// TIA Portal V15.1 export
// export: Created 2024-06-21T08:40:56.5099425Z, ExportSetting WithDefaults, DisplayName Totally Integrated Automation Portal, DisplayVersion V15.1 Update 5, DisplayName TIA Portal Openness, DisplayVersion V15.1 Update 5, DisplayName SINAMICS Startdrive Advanced, DisplayVersion V15.1, DisplayName G130, G150, S120, S150, SINAMICS MV, S210, DisplayVersion V15.1, DisplayName G110M, G120, G120C, G120D, G120P, DisplayVersion V15.1, DisplayName STEP 7 Professional, DisplayVersion V15.1 Update 5, DisplayName STEP 7 Safety, DisplayVersion V15.1, DisplayName WinCC Professional, DisplayVersion V15.1 Update 5, DisplayName SIMATIC Visualization Architect, DisplayVersion V15.1
FUNCTION_BLOCK "L2StopPos"   // FB1310, FBD
TITLE = L2StopPos
{ S7_Optimized_Access := 'TRUE' }
AUTHOR : VCC
FAMILY : Actuator
VERSION : 0.1
// =============================================================================
// This module will be used for a two Position movements.
// It will take care of the Alarms and of the Detections.
// =============================================================================
// stored: AutoNumber false, IsIECCheckEnabled false, IsRetainMemResEnabled false, MemoryReserve 100, SetENOAutomatically False, UDAEnableTagReadback false
   VAR_INPUT
      I_DetSet { ExternalAccessible := 'False'; ExternalVisible := 'False'; ExternalWritable := 'False'} : Bool;   // Set detection signal / Set Detection signal
      I_DetRes { ExternalAccessible := 'False'; ExternalVisible := 'False'; ExternalWritable := 'False'} : Bool;   // Reset detection signal / Reset Detection signal
      I_CmdSet { ExternalAccessible := 'False'; ExternalVisible := 'False'; ExternalWritable := 'False'} : Bool;   // function set command / Function set command
      I_CmdRes { ExternalAccessible := 'False'; ExternalVisible := 'False'; ExternalWritable := 'False'} : Bool;   // Function reset command / Function Reset command
      I_RunSet { ExternalAccessible := 'False'; ExternalVisible := 'False'; ExternalWritable := 'False'} : Bool;   // Memory that the Set function is busy
      I_RunRes { ExternalAccessible := 'False'; ExternalVisible := 'False'; ExternalWritable := 'False'} : Bool;   // Memory that the Reset function is busy
      I_SetIntlkOK { ExternalAccessible := 'False'; ExternalVisible := 'False'; ExternalWritable := 'False'} : Bool := TRUE;   // Set Interlock
      I_ResIntlkOK { ExternalAccessible := 'False'; ExternalVisible := 'False'; ExternalWritable := 'False'} : Bool := TRUE;   // Reset Interlock
      I_SafetyOk { ExternalAccessible := 'False'; ExternalVisible := 'False'; ExternalWritable := 'False'} : Bool;   // Safety Ok
      I_AlarmResetPB { ExternalAccessible := 'False'; ExternalVisible := 'False'; ExternalWritable := 'False'} : Bool := TRUE;   // alarm reset Push Button is activated / Alarm Reset Push Button is Activated
      C_KeepPosition { ExternalAccessible := 'False'; ExternalVisible := 'False'; ExternalWritable := 'False'} : Bool;   // If true, the last position shall be kept ON and checked / If true, the last Position shall be kept ON and checked
      C_EnAlmDet { ExternalAccessible := 'False'; ExternalVisible := 'False'; ExternalWritable := 'False'} : Bool;   // Enable alarm / Enable Alarm
      C_AlarmResetUsed { ExternalAccessible := 'False'; ExternalVisible := 'False'; ExternalWritable := 'False'} : Bool;   // If true, the alarms will be stored untill reseted / If true, the Alarms will be stored untill Reseted
      C_EnAlmOvertime { ExternalAccessible := 'False'; ExternalVisible := 'False'; ExternalWritable := 'False'} : Bool := TRUE;   // Enable Overtime Alarm
      C_ManualClampCmdSet { ExternalAccessible := 'False'; ExternalVisible := 'False'; ExternalWritable := 'False'} : Bool;   // Manual Clamp Set
      C_ManualClampCmdRes { ExternalAccessible := 'False'; ExternalVisible := 'False'; ExternalWritable := 'False'} : Bool;   // Manual Clamp Reset
      C_RunTimeMaxSetWarn { ExternalAccessible := 'False'; ExternalVisible := 'False'; ExternalWritable := 'False'} : DInt;   // Maximum Time (ms) that the function may run (create overtime) / Maximum Time (ms) that the function may run (create Overtime)
      C_RunTimeMaxSetAlm { ExternalAccessible := 'False'; ExternalVisible := 'False'; ExternalWritable := 'False'} : DInt;   // Maximum Time (ms) that the function may run (create overtime) / Maximum Time (ms) that the function may run (create Overtime)
      C_RunTimeMaxResWarn { ExternalAccessible := 'False'; ExternalVisible := 'False'; ExternalWritable := 'False'} : DInt;   // Maximum Time (ms) that the function may run (create overtime) / Maximum Time (ms) that the function may run (create Overtime)
      C_RunTimeMaxResAlm { ExternalAccessible := 'False'; ExternalVisible := 'False'; ExternalWritable := 'False'} : DInt;   // Maximum Time (ms) that the function may run (create overtime) / Maximum Time (ms) that the function may run (create Overtime)
      C_TimeAlmFilt { ExternalAccessible := 'False'; ExternalVisible := 'False'; ExternalWritable := 'False'} : DInt := L#2000;   // timer before any actuator alarm will be active (welding..) / timer before any actuator Alarm will be active (welding..)
      C_AlarmSeverityAB { ExternalAccessible := 'False'; ExternalVisible := 'False'; ExternalWritable := 'False'} : Bool;   // Alarm severity
      C_RunTimeCalculated { ExternalAccessible := 'False'; ExternalVisible := 'False'; ExternalWritable := 'False'} : Bool;   // Maximum Time (ms) that the function may run (create Overtime) is calculated
   END_VAR
   VAR_OUTPUT
      O_SetPos { ExternalAccessible := 'False'; ExternalVisible := 'False'; ExternalWritable := 'False'} : Bool;   // Actuator is in set position / Actuator is in set Position
      O_ResPos { ExternalAccessible := 'False'; ExternalVisible := 'False'; ExternalWritable := 'False'} : Bool;   // Actuator is in reset position / Actuator is in Reset Position
      O_KeepPosSetAlm { ExternalAccessible := 'False'; ExternalVisible := 'False'; ExternalWritable := 'False'} : Bool;   // Detection Set alarm / Detection Set Alarm
      O_KeepPosResAlm { ExternalAccessible := 'False'; ExternalVisible := 'False'; ExternalWritable := 'False'} : Bool;   // Detection Reset alarm / Detection Reset Alarm
      O_TwoDetAlm { ExternalAccessible := 'False'; ExternalVisible := 'False'; ExternalWritable := 'False'} : Bool;   // Fault condition Both detections ON at the same time
      O_OvtSetWarn { ExternalAccessible := 'False'; ExternalVisible := 'False'; ExternalWritable := 'False'} : Bool;   // Warning Overtime Set
      O_OvtResWarn { ExternalAccessible := 'False'; ExternalVisible := 'False'; ExternalWritable := 'False'} : Bool;   // Warning Overtime Reset
      O_OvtSetAlm { ExternalAccessible := 'False'; ExternalVisible := 'False'; ExternalWritable := 'False'} : Bool;   // Alarm Overtime Set
      O_OvtResAlm { ExternalAccessible := 'False'; ExternalVisible := 'False'; ExternalWritable := 'False'} : Bool;   // Alarm Overtime Reset
      O_ConfigCalibrationAlm { ExternalAccessible := 'False'; ExternalVisible := 'False'; ExternalWritable := 'False'} : Bool;   // Alarm Config/Calibration
      O_CalibrationWarn { ExternalAccessible := 'False'; ExternalVisible := 'False'; ExternalWritable := 'False'} : Bool;   // Warning Calibration
      O_AlarmABCondition { ExternalAccessible := 'False'; ExternalVisible := 'False'; ExternalWritable := 'False'} : Bool;   // Alarm AB condition / Alarm AB Condition
      H_IAnim { ExternalAccessible := 'False'; ExternalVisible := 'False'; ExternalWritable := 'False'} : DWord;   // Animation color of icon
   END_VAR
   VAR_IN_OUT
      IO_Modes : "Modes";   // Modes
      H_2StopPos : "H_2StopPos";   // Animation
   END_VAR
   VAR
      AlarmReset { ExternalAccessible := 'False'; ExternalVisible := 'False'; ExternalWritable := 'False'} : Bool;   // Alarm Reset Memory
      SetPosReq { ExternalAccessible := 'False'; ExternalVisible := 'False'; ExternalWritable := 'False'} : Bool;   // Memorisation of the last set movement
      ResPosReq { ExternalAccessible := 'False'; ExternalVisible := 'False'; ExternalWritable := 'False'} : Bool;   // Memorisation of the last reset movement / Memorisation of the last Reset movement
      KeepSetPosOn { ExternalAccessible := 'False'; ExternalVisible := 'False'; ExternalWritable := 'False'} : Bool;   // Check that Set detection is keept on / Check that Set Detection is keept on
      KeepResPosOn { ExternalAccessible := 'False'; ExternalVisible := 'False'; ExternalWritable := 'False'} : Bool;   // Check that Set detection is keept on / Check that Set Detection is keept on
      KeepPosSetStartTimer { ExternalAccessible := 'False'; ExternalVisible := 'False'; ExternalWritable := 'False'} : Bool;   // Detection Set request to start timer / Detection Set Request to start timer
      KeepPosResStartTimer { ExternalAccessible := 'False'; ExternalVisible := 'False'; ExternalWritable := 'False'} : Bool;   // Detection Reset request to start timer / Detection Reset Request to start timer
      TwoDetStartTimer { ExternalAccessible := 'False'; ExternalVisible := 'False'; ExternalWritable := 'False'} : Bool;   // Both detections ON at the same time request to start timer / Both Detections ON at the same time Request to start timer
      AlarmFilterStart { ExternalAccessible := 'False'; ExternalVisible := 'False'; ExternalWritable := 'False'} : Bool;   // Alarm filter must be started
      OvtSetWarnResult { ExternalAccessible := 'False'; ExternalVisible := 'False'; ExternalWritable := 'False'} : Bool;   // Overtime set warning result
      OvtResWarnResult { ExternalAccessible := 'False'; ExternalVisible := 'False'; ExternalWritable := 'False'} : Bool;   // Overtime reset warning result / Overtime Reset warning result
      OvtSetAlmResult { ExternalAccessible := 'False'; ExternalVisible := 'False'; ExternalWritable := 'False'} : Bool;   // Overtime set alarm result / Overtime set Alarm result
      OvtResAlmResult { ExternalAccessible := 'False'; ExternalVisible := 'False'; ExternalWritable := 'False'} : Bool;   // Overtime reset alarm result / Overtime Reset Alarm result
      AlmFilterResult { ExternalAccessible := 'False'; ExternalVisible := 'False'; ExternalWritable := 'False'} : Bool;   // Alarm filter result
      TwoDetAlm { ExternalAccessible := 'False'; ExternalVisible := 'False'; ExternalWritable := 'False'} : Bool;   // Two detection alarm / Set Reset Activated Simultaneously / Set Reset Påverkade Samtidigt
      KeepPosResAlm { ExternalAccessible := 'False'; ExternalVisible := 'False'; ExternalWritable := 'False'} : Bool;   // Keep position Reset alarm / Position Supervision Reset Position / Positionsövervakning Reset Läge
      KeepPosSetAlm { ExternalAccessible := 'False'; ExternalVisible := 'False'; ExternalWritable := 'False'} : Bool;   // Keep position Set alarm / Alarm Keep Position Set Position / Larm Positionsövervakning Set Läge
      OvtResAlm { ExternalAccessible := 'False'; ExternalVisible := 'False'; ExternalWritable := 'False'} : Bool;   // Overtime Reset alarm / Overtime Reset Alarm
      OvtSetAlm { ExternalAccessible := 'False'; ExternalVisible := 'False'; ExternalWritable := 'False'} : Bool;   // Overtime Set alarm / Timeout Set / Tidsövervakning Set
      OvtResWarn { ExternalAccessible := 'False'; ExternalVisible := 'False'; ExternalWritable := 'False'} : Bool;   // Overtime Reset warning
      OvtSetWarn { ExternalAccessible := 'False'; ExternalVisible := 'False'; ExternalWritable := 'False'} : Bool;   // Overtime Set warning
      ConfigCalibrationAlm { ExternalAccessible := 'False'; ExternalVisible := 'False'; ExternalWritable := 'False'} : Bool;   // Config/Calibration Alarm
      CalibrationWarn { ExternalAccessible := 'False'; ExternalVisible := 'False'; ExternalWritable := 'False'} : Bool;   // Warning Calibration
      SetPos { ExternalAccessible := 'False'; ExternalVisible := 'False'; ExternalWritable := 'False'} : Bool;   // Set position / Set Position
      ResPos { ExternalAccessible := 'False'; ExternalVisible := 'False'; ExternalWritable := 'False'} : Bool;   // Reset position / Reset Position
      KeepPosResAlmCond { ExternalAccessible := 'False'; ExternalVisible := 'False'; ExternalWritable := 'False'} : Bool;   // Keep position reset alarm condition / Keep Position Reset Alarm condition
      KeepPosSetAlmCond { ExternalAccessible := 'False'; ExternalVisible := 'False'; ExternalWritable := 'False'} : Bool;   // Keep position set alarm condition / Keep Position Set Alarm condition
      TwoDetAlmCond { ExternalAccessible := 'False'; ExternalVisible := 'False'; ExternalWritable := 'False'} : Bool;   // Two detector alarm condition / Two detector Alarm condition
      OvtResAlmCond { ExternalAccessible := 'False'; ExternalVisible := 'False'; ExternalWritable := 'False'} : Bool;   // Overtime reset alarm condition / Overtime Reset Alarm condition
      OvtSetAlmCond { ExternalAccessible := 'False'; ExternalVisible := 'False'; ExternalWritable := 'False'} : Bool;   // Overtime set alarm condition / Overtime set Alarm condition
      RunSet { ExternalAccessible := 'False'; ExternalVisible := 'False'; ExternalWritable := 'False'} : Bool;   // Memory that the Set function is busy
      RunRes { ExternalAccessible := 'False'; ExternalVisible := 'False'; ExternalWritable := 'False'} : Bool;   // Memory that the Reset function is busy
      Edge { ExternalAccessible := 'False'; ExternalVisible := 'False'; ExternalWritable := 'False'} : Array[1..8] of Bool;   // Edge
      AlarmTimer { ExternalAccessible := 'False'; ExternalVisible := 'False'; ExternalWritable := 'False'} : "LTimer";   // FB
      OvtSetWarnTimer { ExternalAccessible := 'False'; ExternalVisible := 'False'; ExternalWritable := 'False'} : "LTimer";   // FB
      OvtResWarnTimer { ExternalAccessible := 'False'; ExternalVisible := 'False'; ExternalWritable := 'False'} : "LTimer";   // FB
      OvtSetAlmTimer { ExternalAccessible := 'False'; ExternalVisible := 'False'; ExternalWritable := 'False'} : "LTimer";   // FB
      OvtResAlmTimer { ExternalAccessible := 'False'; ExternalVisible := 'False'; ExternalWritable := 'False'} : "LTimer";   // FB
   END_VAR
   VAR RETAIN
      OvtWarnSet { ExternalAccessible := 'False'; ExternalVisible := 'False'; ExternalWritable := 'False'} : DInt;   // Alarm Value
      OvtWarnRes { ExternalAccessible := 'False'; ExternalVisible := 'False'; ExternalWritable := 'False'} : DInt;   // Alarm Value
      OvtAlarmSet { ExternalAccessible := 'False'; ExternalVisible := 'False'; ExternalWritable := 'False'} : DInt;   // Alarm Value
      OvtAlarmRes { ExternalAccessible := 'False'; ExternalVisible := 'False'; ExternalWritable := 'False'} : DInt;   // Alarm Value
      CalibratedSet { ExternalAccessible := 'False'; ExternalVisible := 'False'; ExternalWritable := 'False'} : Bool;   // Calibrated Set
      CalibratedRes { ExternalAccessible := 'False'; ExternalVisible := 'False'; ExternalWritable := 'False'} : Bool;   // Calibrated Reset
   END_VAR
   VAR
      AlarmTimeWithConfig { ExternalAccessible := 'False'; ExternalVisible := 'False'; ExternalWritable := 'False'} : Bool;
      AlarmTimeWithCalibration { ExternalAccessible := 'False'; ExternalVisible := 'False'; ExternalWritable := 'False'} : Bool;
      AlarmTimeWithCalculation { ExternalAccessible := 'False'; ExternalVisible := 'False'; ExternalWritable := 'False'} : Bool;
      AlmFilterTimerValue { ExternalAccessible := 'False'; ExternalVisible := 'False'; ExternalWritable := 'False'} : DInt;
   END_VAR
   VAR_TEMP
      H_CalibrateSet : Bool;   // HMI Function
      H_CalibrateReset : Bool;   // HMI Function
      TempReal : Real;
   END_VAR
   VAR_TEMP   // added for the SCL form of the ladder/FBD networks
      _w1 : Bool;
      _w2 : Bool;
      _w3 : Bool;
      _w4 : Bool;
   END_VAR
BEGIN

REGION Network 1: **** 1 - Inputs **** HMI Commands
   // Extract the Commands from HMIRobCmd / Extract the Commands from HMI
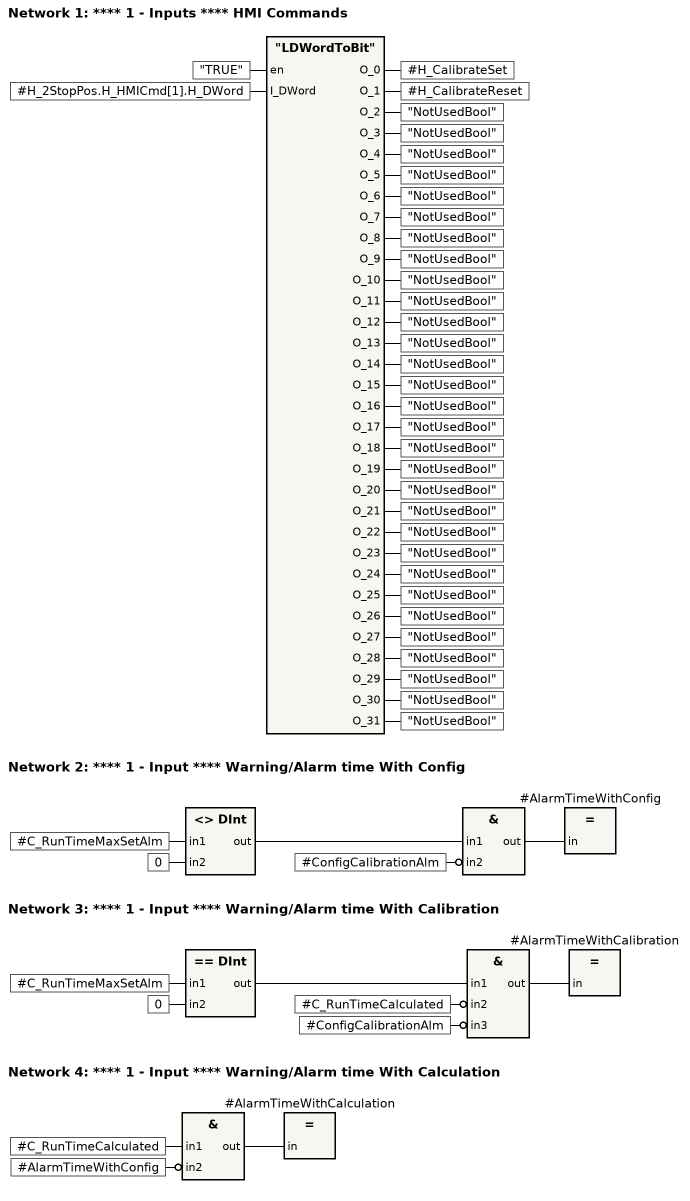
   IF "TRUE" THEN
       "LDWordToBit"(I_DWord := #H_2StopPos.H_HMICmd[1].H_DWord,
                     O_0 => #H_CalibrateSet,
                     O_1 => #H_CalibrateReset,
                     O_2 => "NotUsedBool",
                     O_3 => "NotUsedBool",
                     O_4 => "NotUsedBool",
                     O_5 => "NotUsedBool",
                     O_6 => "NotUsedBool",
                     O_7 => "NotUsedBool",
                     O_8 => "NotUsedBool",
                     O_9 => "NotUsedBool",
                     O_10 => "NotUsedBool",
                     O_11 => "NotUsedBool",
                     O_12 => "NotUsedBool",
                     O_13 => "NotUsedBool",
                     O_14 => "NotUsedBool",
                     O_15 => "NotUsedBool",
                     O_16 => "NotUsedBool",
                     O_17 => "NotUsedBool",
                     O_18 => "NotUsedBool",
                     O_19 => "NotUsedBool",
                     O_20 => "NotUsedBool",
                     O_21 => "NotUsedBool",
                     O_22 => "NotUsedBool",
                     O_23 => "NotUsedBool",
                     O_24 => "NotUsedBool",
                     O_25 => "NotUsedBool",
                     O_26 => "NotUsedBool",
                     O_27 => "NotUsedBool",
                     O_28 => "NotUsedBool",
                     O_29 => "NotUsedBool",
                     O_30 => "NotUsedBool",
                     O_31 => "NotUsedBool");
   END_IF;
END_REGION

REGION Network 2: **** 1 - Input **** Warning/Alarm time With Config
   #AlarmTimeWithConfig := (#C_RunTimeMaxSetAlm <> 0) AND NOT #ConfigCalibrationAlm;
END_REGION

REGION Network 3: **** 1 - Input **** Warning/Alarm time With Calibration
   #AlarmTimeWithCalibration := (#C_RunTimeMaxSetAlm = 0) AND NOT #C_RunTimeCalculated AND NOT #ConfigCalibrationAlm;
END_REGION

REGION Network 4: **** 1 - Input **** Warning/Alarm time With Calculation
   #AlarmTimeWithCalculation := #C_RunTimeCalculated AND NOT #AlarmTimeWithConfig;
END_REGION

REGION Network 5: Calibrated Set / **** 1 - Input **** Ovt Values / **** 1 - Inputs **** Ovt Values
   // Ovt Values
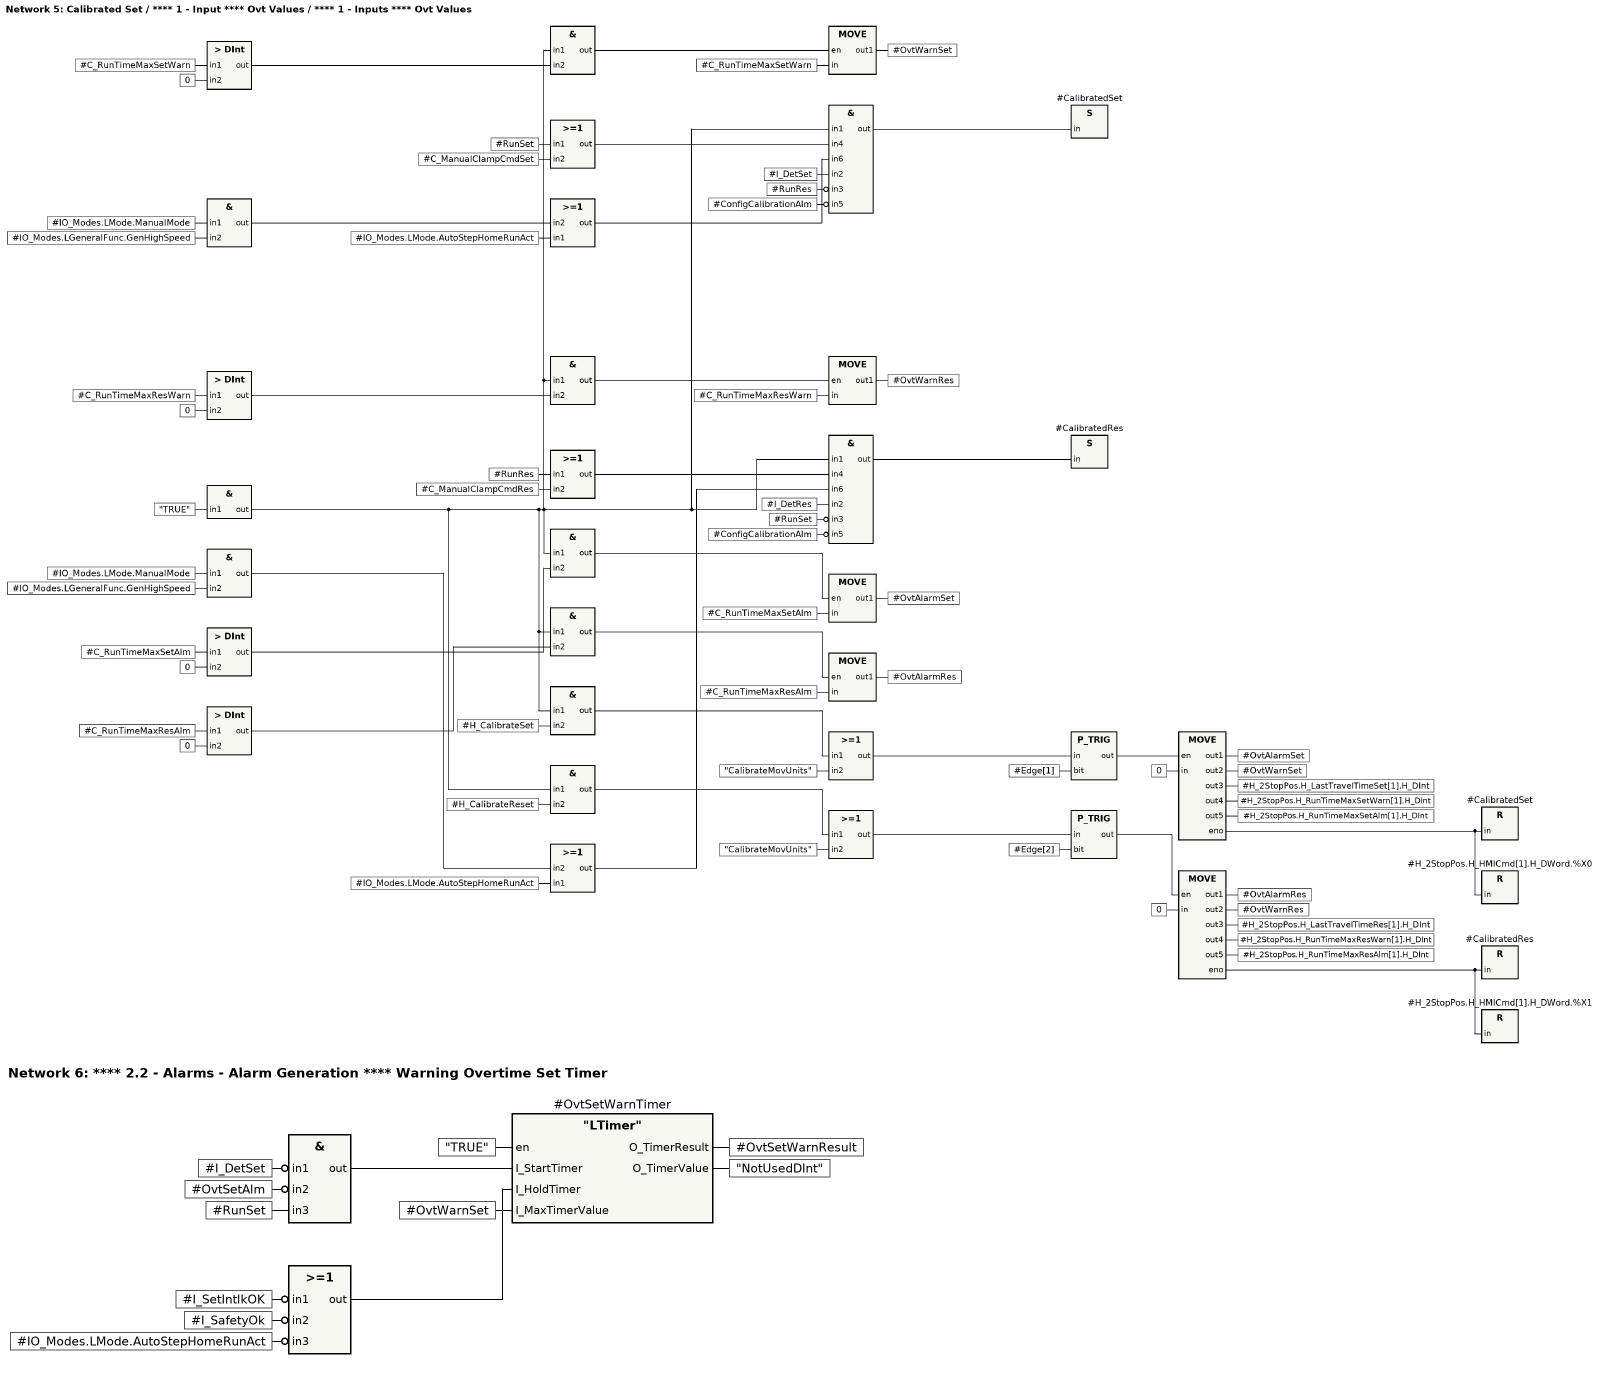
   // ENO of a box is taken as its EN; it also drops when the box reports an error
   IF "TRUE" AND (#C_RunTimeMaxSetWarn > 0) THEN #OvtWarnSet := #C_RunTimeMaxSetWarn; END_IF;
   IF "TRUE" AND (#C_RunTimeMaxResWarn > 0) THEN #OvtWarnRes := #C_RunTimeMaxResWarn; END_IF;
   IF "TRUE" AND (#C_RunTimeMaxSetAlm > 0) THEN #OvtAlarmSet := #C_RunTimeMaxSetAlm; END_IF;
   IF "TRUE" AND (#C_RunTimeMaxResAlm > 0) THEN #OvtAlarmRes := #C_RunTimeMaxResAlm; END_IF;
   IF "TRUE" AND (#RunSet OR #C_ManualClampCmdSet) AND ((#IO_Modes.LMode.ManualMode AND #IO_Modes.LGeneralFunc.GenHighSpeed) OR #IO_Modes.LMode.AutoStepHomeRunAct) AND #I_DetSet AND NOT #RunRes AND NOT #ConfigCalibrationAlm THEN
       #CalibratedSet := TRUE;
   END_IF;
   IF "TRUE" AND (#RunRes OR #C_ManualClampCmdRes) AND ((#IO_Modes.LMode.ManualMode AND #IO_Modes.LGeneralFunc.GenHighSpeed) OR #IO_Modes.LMode.AutoStepHomeRunAct) AND #I_DetRes AND NOT #RunSet AND NOT #ConfigCalibrationAlm THEN
       #CalibratedRes := TRUE;
   END_IF;
   #_w1 := ("TRUE" AND #H_CalibrateSet) OR "CalibrateMovUnits";
   #_w2 := #_w1 AND NOT #Edge[1];   // rising edge
   #Edge[1] := #_w1;
   IF #_w2 THEN
       #OvtAlarmSet := 0;
       #OvtWarnSet := 0;
       #H_2StopPos.H_LastTravelTimeSet[1].H_DInt := 0;
       #H_2StopPos.H_RunTimeMaxSetWarn[1].H_DInt := 0;
       #H_2StopPos.H_RunTimeMaxSetAlm[1].H_DInt := 0;
       #CalibratedSet := FALSE;
       #H_2StopPos.H_HMICmd[1].H_DWord.%X0 := FALSE;
   END_IF;
   #_w3 := ("TRUE" AND #H_CalibrateReset) OR "CalibrateMovUnits";
   #_w4 := #_w3 AND NOT #Edge[2];   // rising edge
   #Edge[2] := #_w3;
   IF #_w4 THEN
       #OvtAlarmRes := 0;
       #OvtWarnRes := 0;
       #H_2StopPos.H_LastTravelTimeRes[1].H_DInt := 0;
       #H_2StopPos.H_RunTimeMaxResWarn[1].H_DInt := 0;
       #H_2StopPos.H_RunTimeMaxResAlm[1].H_DInt := 0;
       #CalibratedRes := FALSE;
       #H_2StopPos.H_HMICmd[1].H_DWord.%X1 := FALSE;
   END_IF;
END_REGION

REGION Network 6: **** 2.2 - Alarms - Alarm Generation **** Warning Overtime Set Timer
   // Warning Overtime Set Timer
   IF "TRUE" THEN
       #OvtSetWarnTimer(I_StartTimer := NOT #I_DetSet AND NOT #OvtSetAlm AND #RunSet,   // "LTimer"
                        I_HoldTimer := NOT #I_SetIntlkOK OR NOT #I_SafetyOk OR NOT #IO_Modes.LMode.AutoStepHomeRunAct,
                        I_MaxTimerValue := #OvtWarnSet,
                        O_TimerResult => #OvtSetWarnResult,
                        O_TimerValue => "NotUsedDInt");
   END_IF;
END_REGION

REGION Network 7: **** 2.2 - Alarms - Alarm Generation **** Warning Overtime Set Memorisation
   // Warning Overtime Set Memorisation
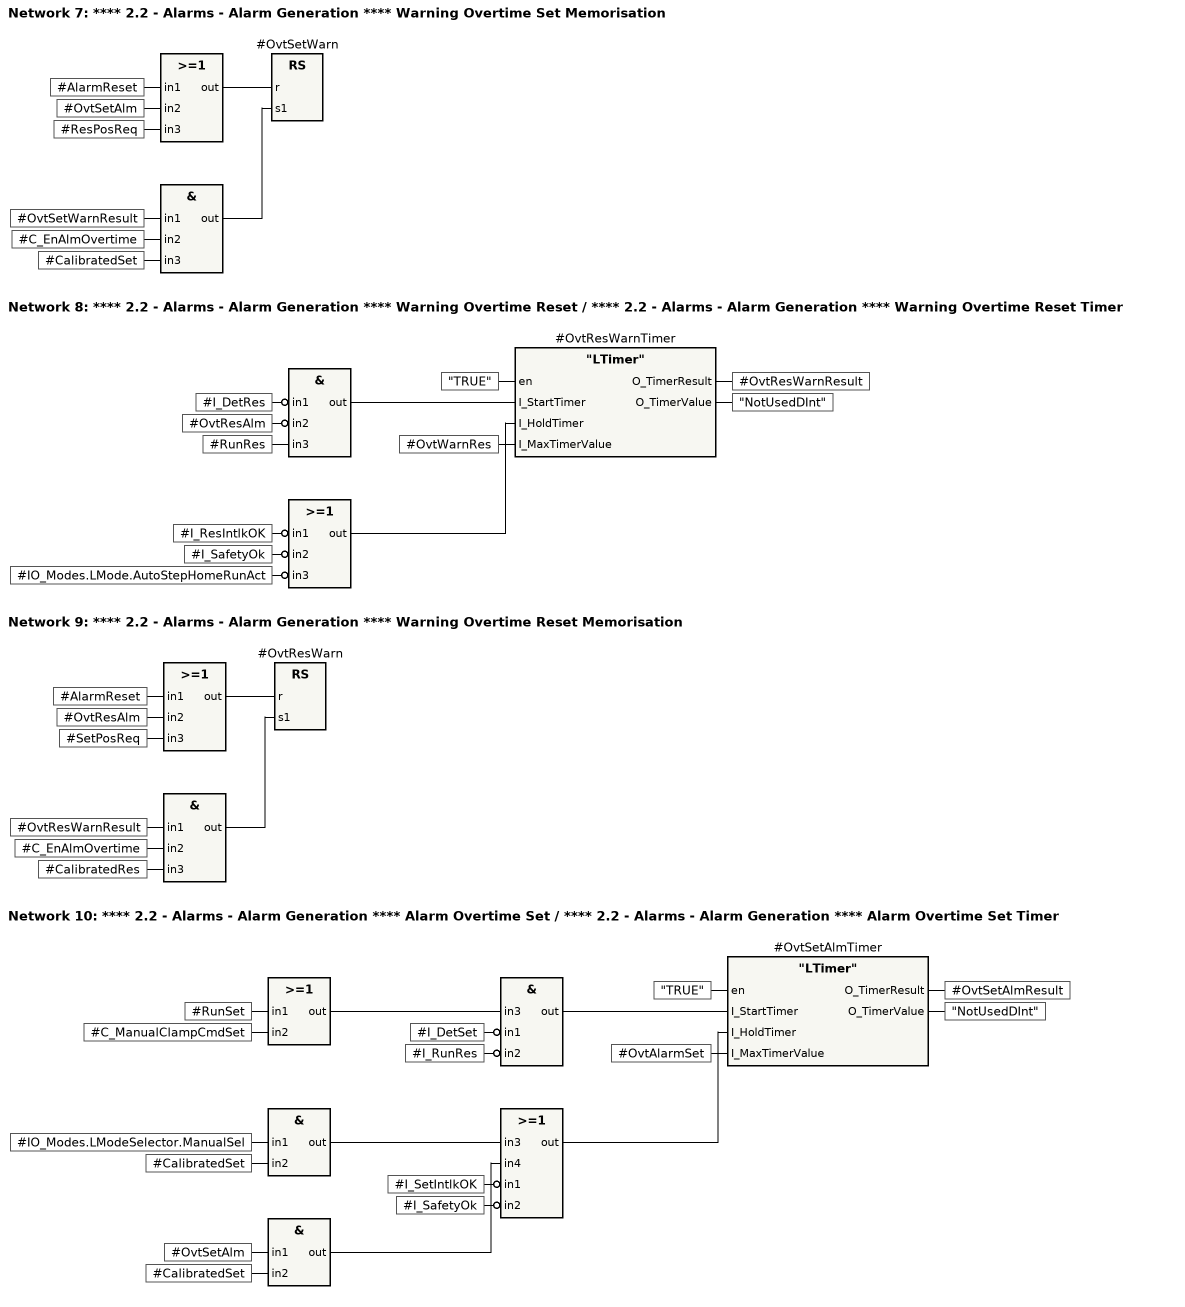
   IF #AlarmReset OR #OvtSetAlm OR #ResPosReq THEN
       #OvtSetWarn := FALSE;   // RS flip-flop
   END_IF;
   IF #OvtSetWarnResult AND #C_EnAlmOvertime AND #CalibratedSet THEN #OvtSetWarn := TRUE; END_IF;
END_REGION

REGION Network 8: **** 2.2 - Alarms - Alarm Generation **** Warning Overtime Reset / **** 2.2 - Alarms - Alarm Generation **** Warning Overtime Reset Timer
   // Warning Overtime Reset
   IF "TRUE" THEN
       #OvtResWarnTimer(I_StartTimer := NOT #I_DetRes AND NOT #OvtResAlm AND #RunRes,   // "LTimer"
                        I_HoldTimer := NOT #I_ResIntlkOK OR NOT #I_SafetyOk OR NOT #IO_Modes.LMode.AutoStepHomeRunAct,
                        I_MaxTimerValue := #OvtWarnRes,
                        O_TimerResult => #OvtResWarnResult,
                        O_TimerValue => "NotUsedDInt");
   END_IF;
END_REGION

REGION Network 9: **** 2.2 - Alarms - Alarm Generation **** Warning Overtime Reset Memorisation
   // Warning Overtime Reset  Memorisation
   IF #AlarmReset OR #OvtResAlm OR #SetPosReq THEN
       #OvtResWarn := FALSE;   // RS flip-flop
   END_IF;
   IF #OvtResWarnResult AND #C_EnAlmOvertime AND #CalibratedRes THEN #OvtResWarn := TRUE; END_IF;
END_REGION

REGION Network 10: **** 2.2 - Alarms - Alarm Generation **** Alarm Overtime Set / **** 2.2 - Alarms - Alarm Generation **** Alarm Overtime Set Timer
   // Alarm Overtime Set
   IF "TRUE" THEN
       #OvtSetAlmTimer(I_StartTimer := (#RunSet OR #C_ManualClampCmdSet) AND NOT #I_DetSet AND NOT #I_RunRes,   // "LTimer"
                       I_HoldTimer := (#IO_Modes.LModeSelector.ManualSel AND #CalibratedSet) OR (#OvtSetAlm AND #CalibratedSet) OR NOT #I_SetIntlkOK OR NOT #I_SafetyOk,
                       I_MaxTimerValue := #OvtAlarmSet,
                       O_TimerResult => #OvtSetAlmResult,
                       O_TimerValue => "NotUsedDInt");
   END_IF;
END_REGION

REGION Network 11: **** 2.2 - Alarms - Alarm Generation **** Alarm Overtime Set Timer -- Calculation Warning/Alarm Time
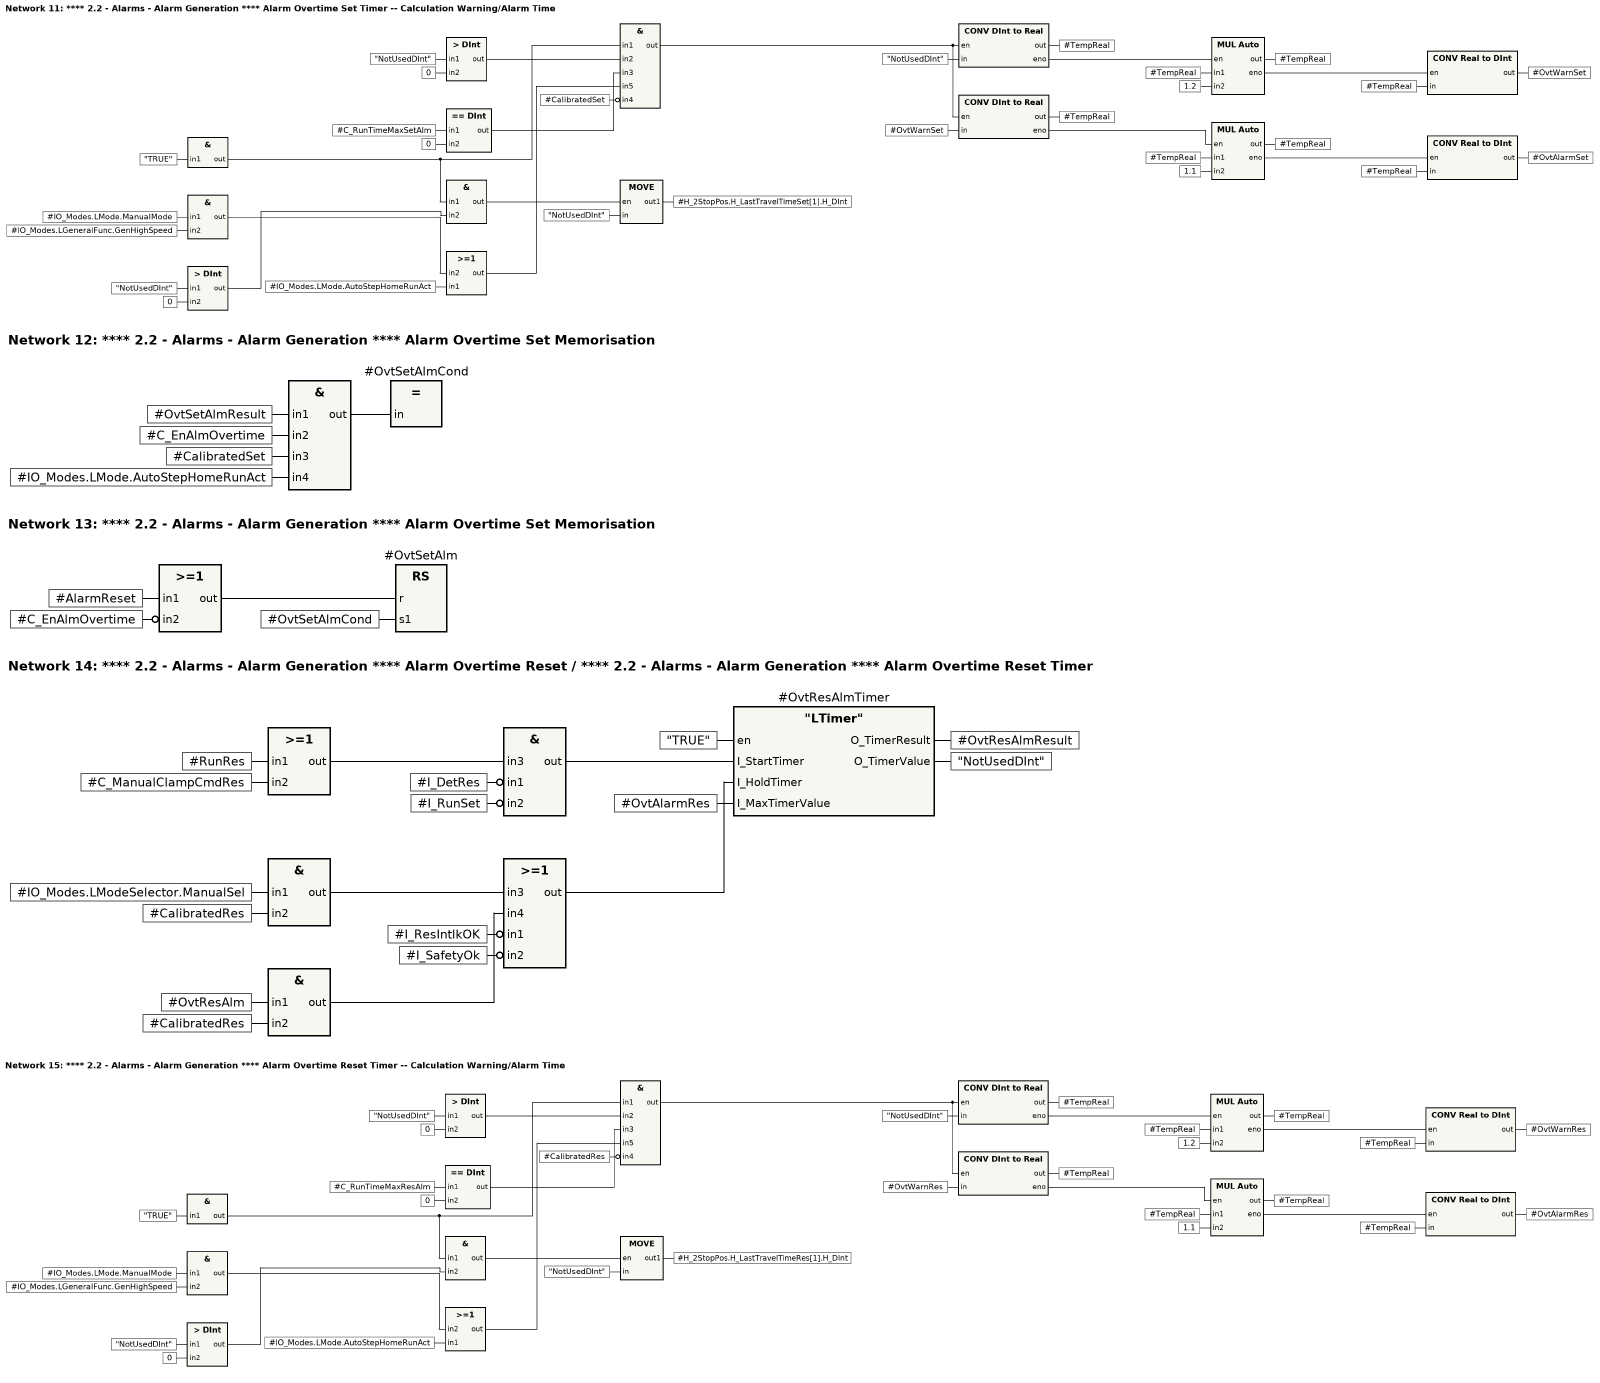
   IF "TRUE" AND ("NotUsedDInt" > 0) AND (#C_RunTimeMaxSetAlm = 0) AND ((#IO_Modes.LMode.ManualMode AND #IO_Modes.LGeneralFunc.GenHighSpeed) OR #IO_Modes.LMode.AutoStepHomeRunAct) AND NOT #CalibratedSet THEN
       #TempReal := DINT_TO_REAL("NotUsedDInt");
       #TempReal := #TempReal * 1.2;
       #OvtWarnSet := REAL_TO_DINT(#TempReal);
       #TempReal := DINT_TO_REAL(#OvtWarnSet);
       #TempReal := #TempReal * 1.1;
       #OvtAlarmSet := REAL_TO_DINT(#TempReal);
   END_IF;
   IF "TRUE" AND ("NotUsedDInt" > 0) THEN #H_2StopPos.H_LastTravelTimeSet[1].H_DInt := "NotUsedDInt"; END_IF;
END_REGION

REGION Network 12: **** 2.2 - Alarms - Alarm Generation **** Alarm Overtime Set Memorisation
   // Alarm Overtime Set Memorisation
   #OvtSetAlmCond := #OvtSetAlmResult AND #C_EnAlmOvertime AND #CalibratedSet AND #IO_Modes.LMode.AutoStepHomeRunAct;
END_REGION

REGION Network 13: **** 2.2 - Alarms - Alarm Generation **** Alarm Overtime Set Memorisation
   // Alarm Overtime Set Memorisation
   IF #AlarmReset OR NOT #C_EnAlmOvertime THEN
       #OvtSetAlm := FALSE;   // RS flip-flop
   END_IF;
   IF #OvtSetAlmCond THEN #OvtSetAlm := TRUE; END_IF;
END_REGION

REGION Network 14: **** 2.2 - Alarms - Alarm Generation **** Alarm Overtime Reset / **** 2.2 - Alarms - Alarm Generation **** Alarm Overtime Reset Timer
   // Alarm Overtime Reset
   IF "TRUE" THEN
       #OvtResAlmTimer(I_StartTimer := (#RunRes OR #C_ManualClampCmdRes) AND NOT #I_DetRes AND NOT #I_RunSet,   // "LTimer"
                       I_HoldTimer := (#IO_Modes.LModeSelector.ManualSel AND #CalibratedRes) OR (#OvtResAlm AND #CalibratedRes) OR NOT #I_ResIntlkOK OR NOT #I_SafetyOk,
                       I_MaxTimerValue := #OvtAlarmRes,
                       O_TimerResult => #OvtResAlmResult,
                       O_TimerValue => "NotUsedDInt");
   END_IF;
END_REGION

REGION Network 15: **** 2.2 - Alarms - Alarm Generation **** Alarm Overtime Reset Timer -- Calculation Warning/Alarm Time
   IF "TRUE" AND ("NotUsedDInt" > 0) AND (#C_RunTimeMaxResAlm = 0) AND ((#IO_Modes.LMode.ManualMode AND #IO_Modes.LGeneralFunc.GenHighSpeed) OR #IO_Modes.LMode.AutoStepHomeRunAct) AND NOT #CalibratedRes THEN
       #TempReal := DINT_TO_REAL("NotUsedDInt");
       #TempReal := #TempReal * 1.2;
       #OvtWarnRes := REAL_TO_DINT(#TempReal);
       #TempReal := DINT_TO_REAL(#OvtWarnRes);
       #TempReal := #TempReal * 1.1;
       #OvtAlarmRes := REAL_TO_DINT(#TempReal);
   END_IF;
   IF "TRUE" AND ("NotUsedDInt" > 0) THEN #H_2StopPos.H_LastTravelTimeRes[1].H_DInt := "NotUsedDInt"; END_IF;
END_REGION

REGION Network 16: **** 2.2 - Alarms - Alarm Generation **** Alarm Overtime Reset Memorisation
   // Alarm Overtime Reset  Memorisation
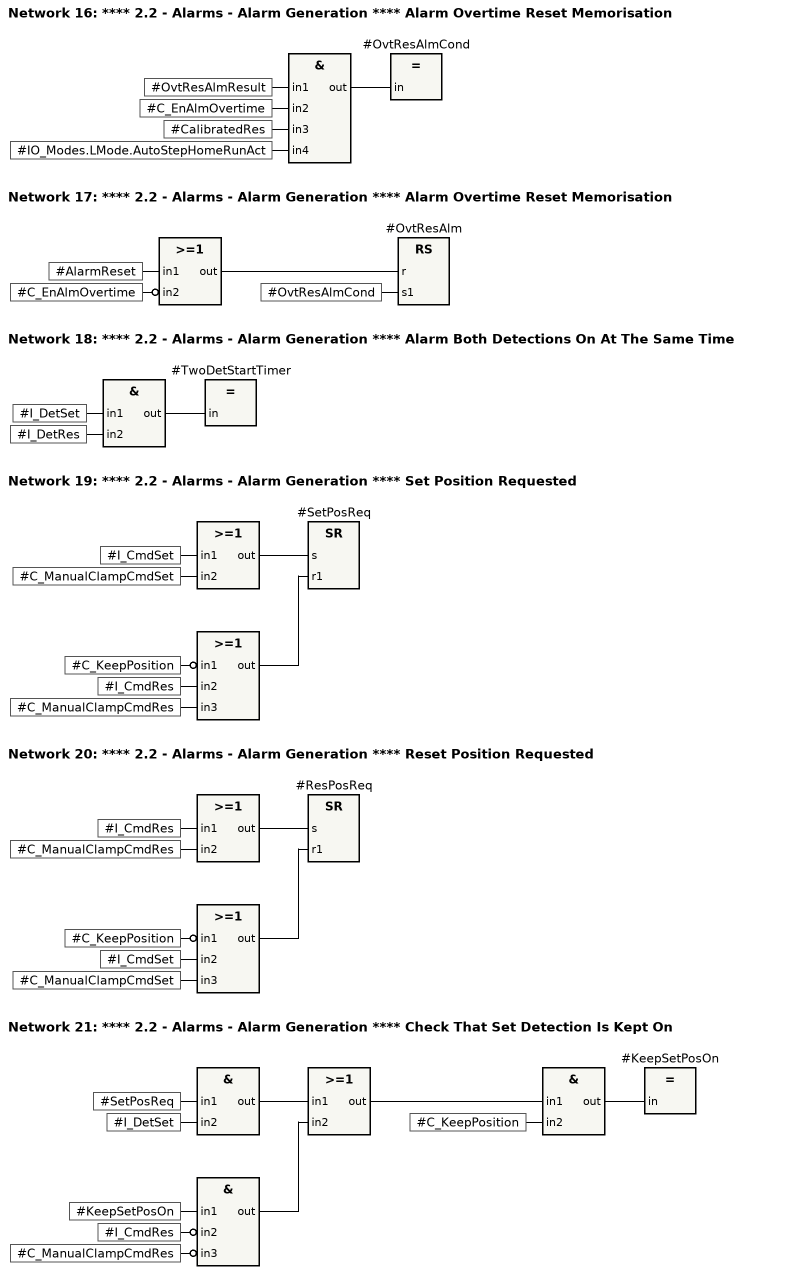
   #OvtResAlmCond := #OvtResAlmResult AND #C_EnAlmOvertime AND #CalibratedRes AND #IO_Modes.LMode.AutoStepHomeRunAct;
END_REGION

REGION Network 17: **** 2.2 - Alarms - Alarm Generation **** Alarm Overtime Reset Memorisation
   // Alarm Overtime Reset  Memorisation
   IF #AlarmReset OR NOT #C_EnAlmOvertime THEN
       #OvtResAlm := FALSE;   // RS flip-flop
   END_IF;
   IF #OvtResAlmCond THEN #OvtResAlm := TRUE; END_IF;
END_REGION

REGION Network 18: **** 2.2 - Alarms - Alarm Generation **** Alarm Both Detections On At The Same Time
   // Alarm Both Detections On At The Same Time
   #TwoDetStartTimer := #I_DetSet AND #I_DetRes;
END_REGION

REGION Network 19: **** 2.2 - Alarms - Alarm Generation **** Set Position Requested
   // Set Position Requested
   IF #I_CmdSet OR #C_ManualClampCmdSet THEN
       #SetPosReq := TRUE;   // SR flip-flop
   END_IF;
   IF NOT #C_KeepPosition OR #I_CmdRes OR #C_ManualClampCmdRes THEN #SetPosReq := FALSE; END_IF;
END_REGION

REGION Network 20: **** 2.2 - Alarms - Alarm Generation **** Reset Position Requested
   // Reset  Position Requested
   IF #I_CmdRes OR #C_ManualClampCmdRes THEN
       #ResPosReq := TRUE;   // SR flip-flop
   END_IF;
   IF NOT #C_KeepPosition OR #I_CmdSet OR #C_ManualClampCmdSet THEN #ResPosReq := FALSE; END_IF;
END_REGION

REGION Network 21: **** 2.2 - Alarms - Alarm Generation **** Check That Set Detection Is Kept On
   // Check That Set Detection Is Kept On
   #KeepSetPosOn := ((#SetPosReq AND #I_DetSet) OR (#KeepSetPosOn AND NOT #I_CmdRes AND NOT #C_ManualClampCmdRes)) AND #C_KeepPosition;
END_REGION

REGION Network 22: **** 2.2 - Alarms - Alarm Generation **** Check That Reset Detection Is Kept On
   // Check That Reset  Detection Is Kept On
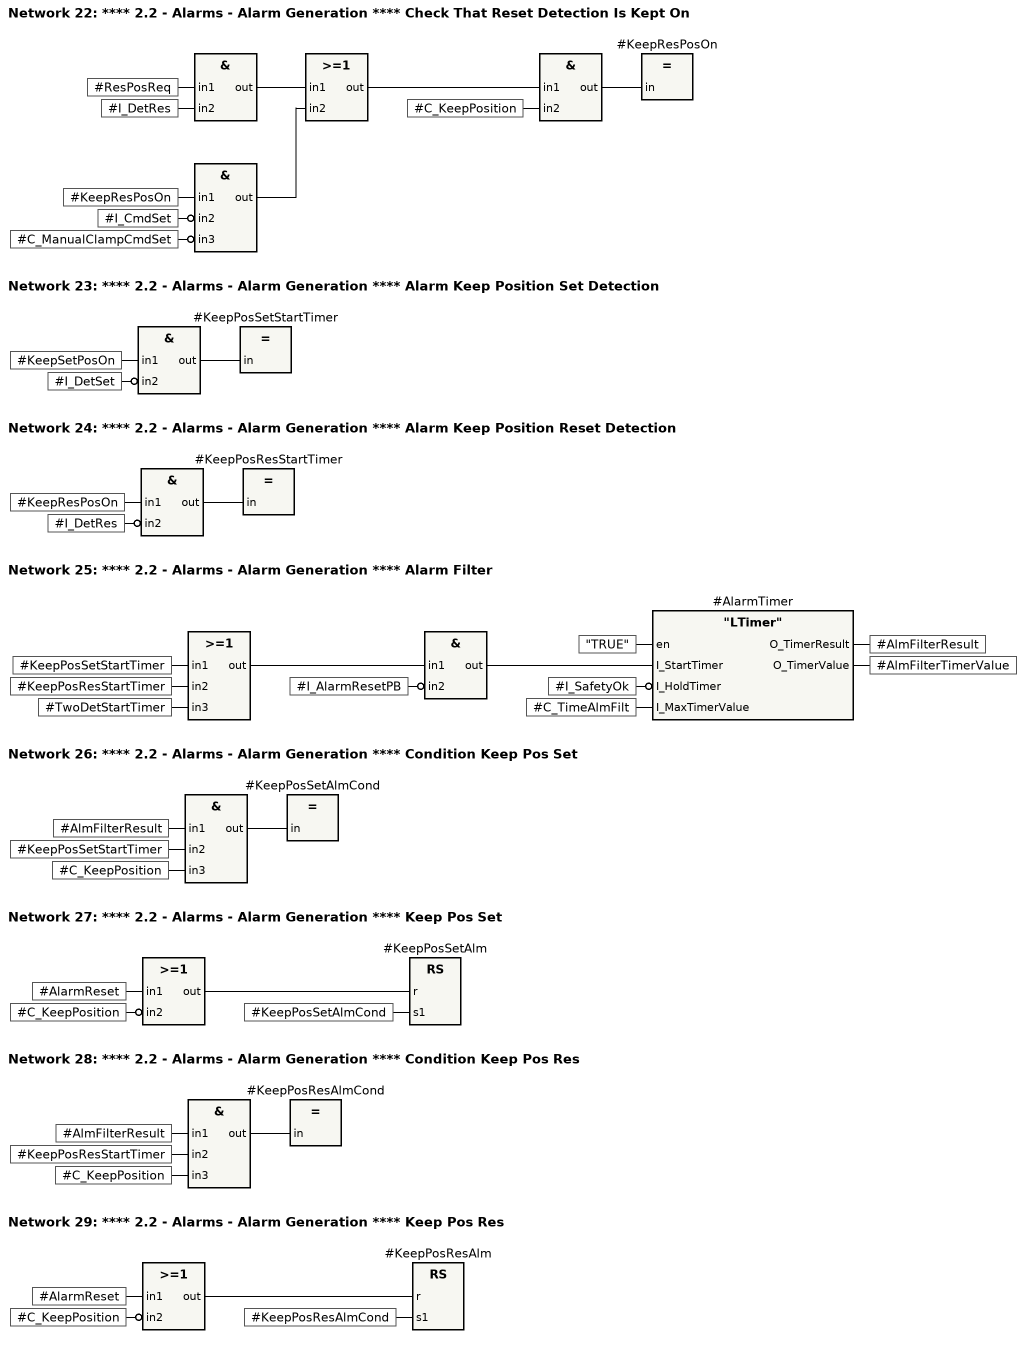
   #KeepResPosOn := ((#ResPosReq AND #I_DetRes) OR (#KeepResPosOn AND NOT #I_CmdSet AND NOT #C_ManualClampCmdSet)) AND #C_KeepPosition;
END_REGION

REGION Network 23: **** 2.2 - Alarms - Alarm Generation **** Alarm Keep Position Set Detection
   // Alarm keep Position Set Detection
   #KeepPosSetStartTimer := #KeepSetPosOn AND NOT #I_DetSet;
END_REGION

REGION Network 24: **** 2.2 - Alarms - Alarm Generation **** Alarm Keep Position Reset Detection
   // Alarm Keep Position Reset  Detection
   #KeepPosResStartTimer := #KeepResPosOn AND NOT #I_DetRes;
END_REGION

REGION Network 25: **** 2.2 - Alarms - Alarm Generation **** Alarm Filter
   // Alarm Filter
   IF "TRUE" THEN
       #AlarmTimer(I_StartTimer := (#KeepPosSetStartTimer OR #KeepPosResStartTimer OR #TwoDetStartTimer) AND NOT #I_AlarmResetPB,   // "LTimer"
                   I_HoldTimer := NOT #I_SafetyOk,
                   I_MaxTimerValue := #C_TimeAlmFilt,
                   O_TimerResult => #AlmFilterResult,
                   O_TimerValue => #AlmFilterTimerValue);
   END_IF;
END_REGION

REGION Network 26: **** 2.2 - Alarms - Alarm Generation **** Condition Keep Pos Set
   // Condition Keep Pos Set
   #KeepPosSetAlmCond := #AlmFilterResult AND #KeepPosSetStartTimer AND #C_KeepPosition;
END_REGION

REGION Network 27: **** 2.2 - Alarms - Alarm Generation **** Keep Pos Set
   // Keep Pos Set
   IF #AlarmReset OR NOT #C_KeepPosition THEN
       #KeepPosSetAlm := FALSE;   // RS flip-flop
   END_IF;
   IF #KeepPosSetAlmCond THEN #KeepPosSetAlm := TRUE; END_IF;
END_REGION

REGION Network 28: **** 2.2 - Alarms - Alarm Generation **** Condition Keep Pos Res
   // Condition Keep Pos Res
   #KeepPosResAlmCond := #AlmFilterResult AND #KeepPosResStartTimer AND #C_KeepPosition;
END_REGION

REGION Network 29: **** 2.2 - Alarms - Alarm Generation **** Keep Pos Res
   // Keep Pos Res
   IF #AlarmReset OR NOT #C_KeepPosition THEN
       #KeepPosResAlm := FALSE;   // RS flip-flop
   END_IF;
   IF #KeepPosResAlmCond THEN #KeepPosResAlm := TRUE; END_IF;
END_REGION

REGION Network 30: **** 2.2 - Alarms - Alarm Generation **** 2 Detection Alarm
   // 2 Detection Alarm
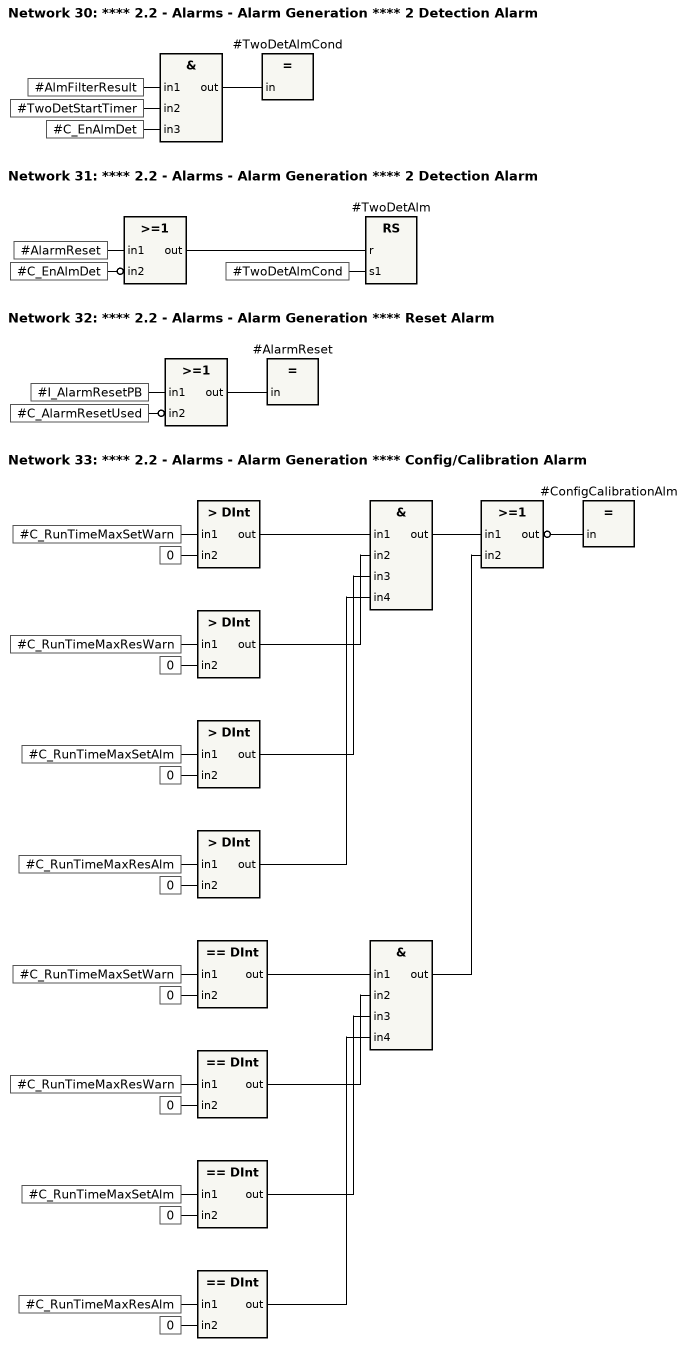
   #TwoDetAlmCond := #AlmFilterResult AND #TwoDetStartTimer AND #C_EnAlmDet;
END_REGION

REGION Network 31: **** 2.2 - Alarms - Alarm Generation **** 2 Detection Alarm
   // 2 Detection Alarm
   IF #AlarmReset OR NOT #C_EnAlmDet THEN
       #TwoDetAlm := FALSE;   // RS flip-flop
   END_IF;
   IF #TwoDetAlmCond THEN #TwoDetAlm := TRUE; END_IF;
END_REGION

REGION Network 32: **** 2.2 - Alarms - Alarm Generation **** Reset Alarm
   // Reset  Alarm
   #AlarmReset := #I_AlarmResetPB OR NOT #C_AlarmResetUsed;
END_REGION

REGION Network 33: **** 2.2 - Alarms - Alarm Generation **** Config/Calibration Alarm
   #ConfigCalibrationAlm := NOT (((#C_RunTimeMaxSetWarn > 0) AND (#C_RunTimeMaxResWarn > 0) AND (#C_RunTimeMaxSetAlm > 0) AND (#C_RunTimeMaxResAlm > 0)) OR ((#C_RunTimeMaxSetWarn = 0) AND (#C_RunTimeMaxResWarn = 0) AND (#C_RunTimeMaxSetAlm = 0) AND (#C_RunTimeMaxResAlm = 0)));
END_REGION

REGION Network 34: **** 2.2 - Alarms - Alarm Generation **** Calibration Warning
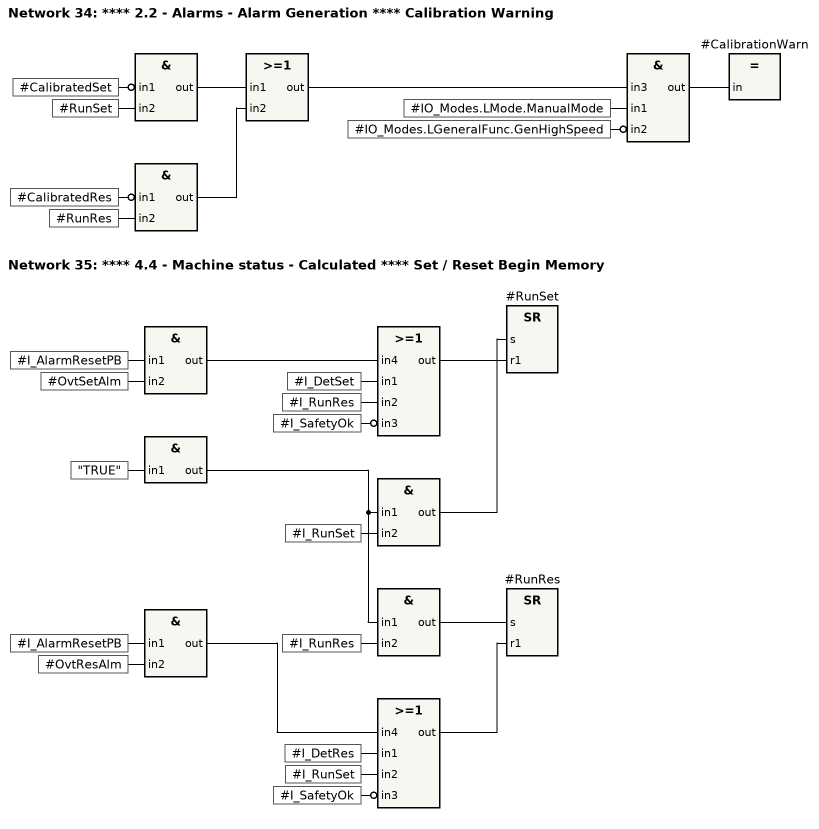
   #CalibrationWarn := ((NOT #CalibratedSet AND #RunSet) OR (NOT #CalibratedRes AND #RunRes)) AND #IO_Modes.LMode.ManualMode AND NOT #IO_Modes.LGeneralFunc.GenHighSpeed;
END_REGION

REGION Network 35: **** 4.4 - Machine status - Calculated **** Set / Reset Begin Memory
   // Set / Reset Begin Memory / Delay of Set Position
   IF "TRUE" AND #I_RunSet THEN
       #RunSet := TRUE;   // SR flip-flop
   END_IF;
   IF (#I_AlarmResetPB AND #OvtSetAlm) OR #I_DetSet OR #I_RunRes OR NOT #I_SafetyOk THEN
       #RunSet := FALSE;
   END_IF;
   IF "TRUE" AND #I_RunRes THEN
       #RunRes := TRUE;   // SR flip-flop
   END_IF;
   IF (#I_AlarmResetPB AND #OvtResAlm) OR #I_DetRes OR #I_RunSet OR NOT #I_SafetyOk THEN
       #RunRes := FALSE;
   END_IF;
END_REGION

REGION Network 36: **** 4.6 - Machine Status - Indication **** Icon Animation / **** 4.6 - Machine status - Indication **** Icon Animation
   // Icon Animation
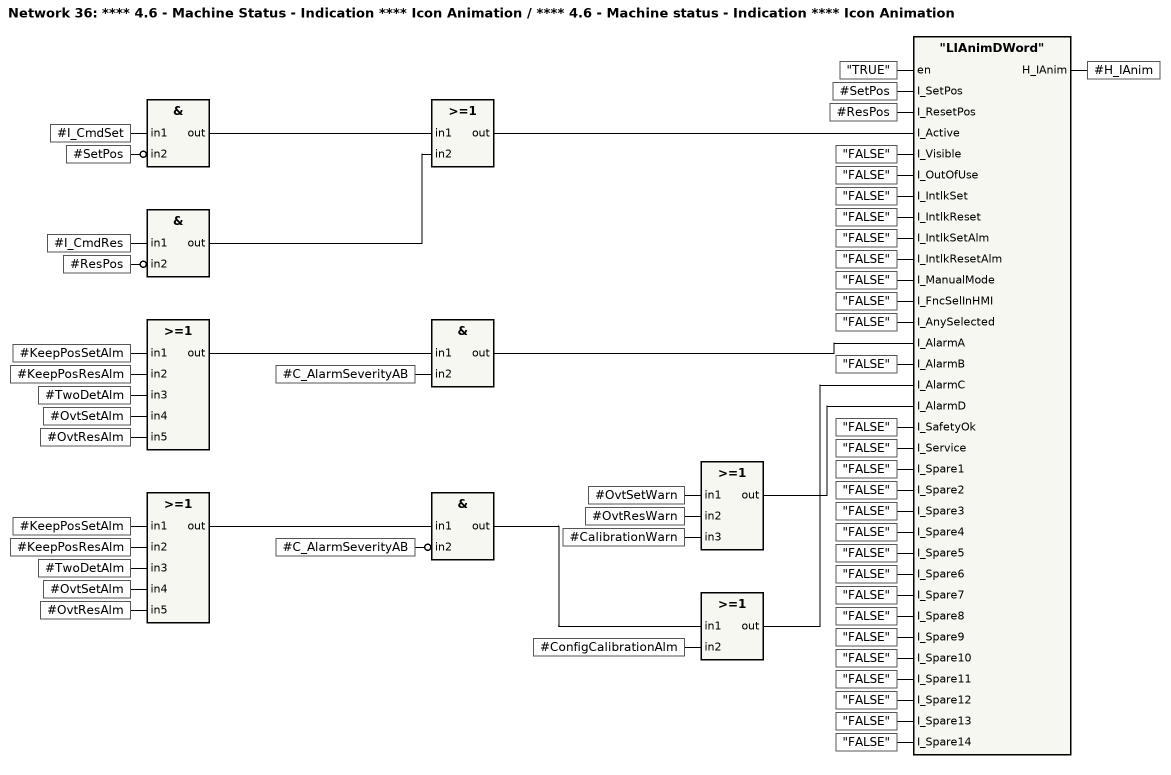
   IF "TRUE" THEN
       "LIAnimDWord"(I_SetPos := #SetPos,
                     I_ResetPos := #ResPos,
                     I_Active := (#I_CmdSet AND NOT #SetPos) OR (#I_CmdRes AND NOT #ResPos),
                     I_Visible := "FALSE",
                     I_OutOfUse := "FALSE",
                     I_IntlkSet := "FALSE",
                     I_IntlkReset := "FALSE",
                     I_IntlkSetAlm := "FALSE",
                     I_IntlkResetAlm := "FALSE",
                     I_ManualMode := "FALSE",
                     I_FncSelInHMI := "FALSE",
                     I_AnySelected := "FALSE",
                     I_AlarmA := (#KeepPosSetAlm OR #KeepPosResAlm OR #TwoDetAlm OR #OvtSetAlm OR #OvtResAlm) AND #C_AlarmSeverityAB,
                     I_AlarmB := "FALSE",
                     I_AlarmC := ((#KeepPosSetAlm OR #KeepPosResAlm OR #TwoDetAlm OR #OvtSetAlm OR #OvtResAlm) AND NOT #C_AlarmSeverityAB) OR #ConfigCalibrationAlm,
                     I_AlarmD := #OvtSetWarn OR #OvtResWarn OR #CalibrationWarn,
                     I_SafetyOk := "FALSE",
                     I_Service := "FALSE",
                     I_Spare1 := "FALSE",
                     I_Spare2 := "FALSE",
                     I_Spare3 := "FALSE",
                     I_Spare4 := "FALSE",
                     I_Spare5 := "FALSE",
                     I_Spare6 := "FALSE",
                     I_Spare7 := "FALSE",
                     I_Spare8 := "FALSE",
                     I_Spare9 := "FALSE",
                     I_Spare10 := "FALSE",
                     I_Spare11 := "FALSE",
                     I_Spare12 := "FALSE",
                     I_Spare13 := "FALSE",
                     I_Spare14 := "FALSE",
                     H_IAnim => #H_IAnim);
   END_IF;
END_REGION

REGION Network 37: **** 4.6 - Machine Status - Indication **** Animation / **** 4.6 - Machine status - Indication **** Animation
   // Animation
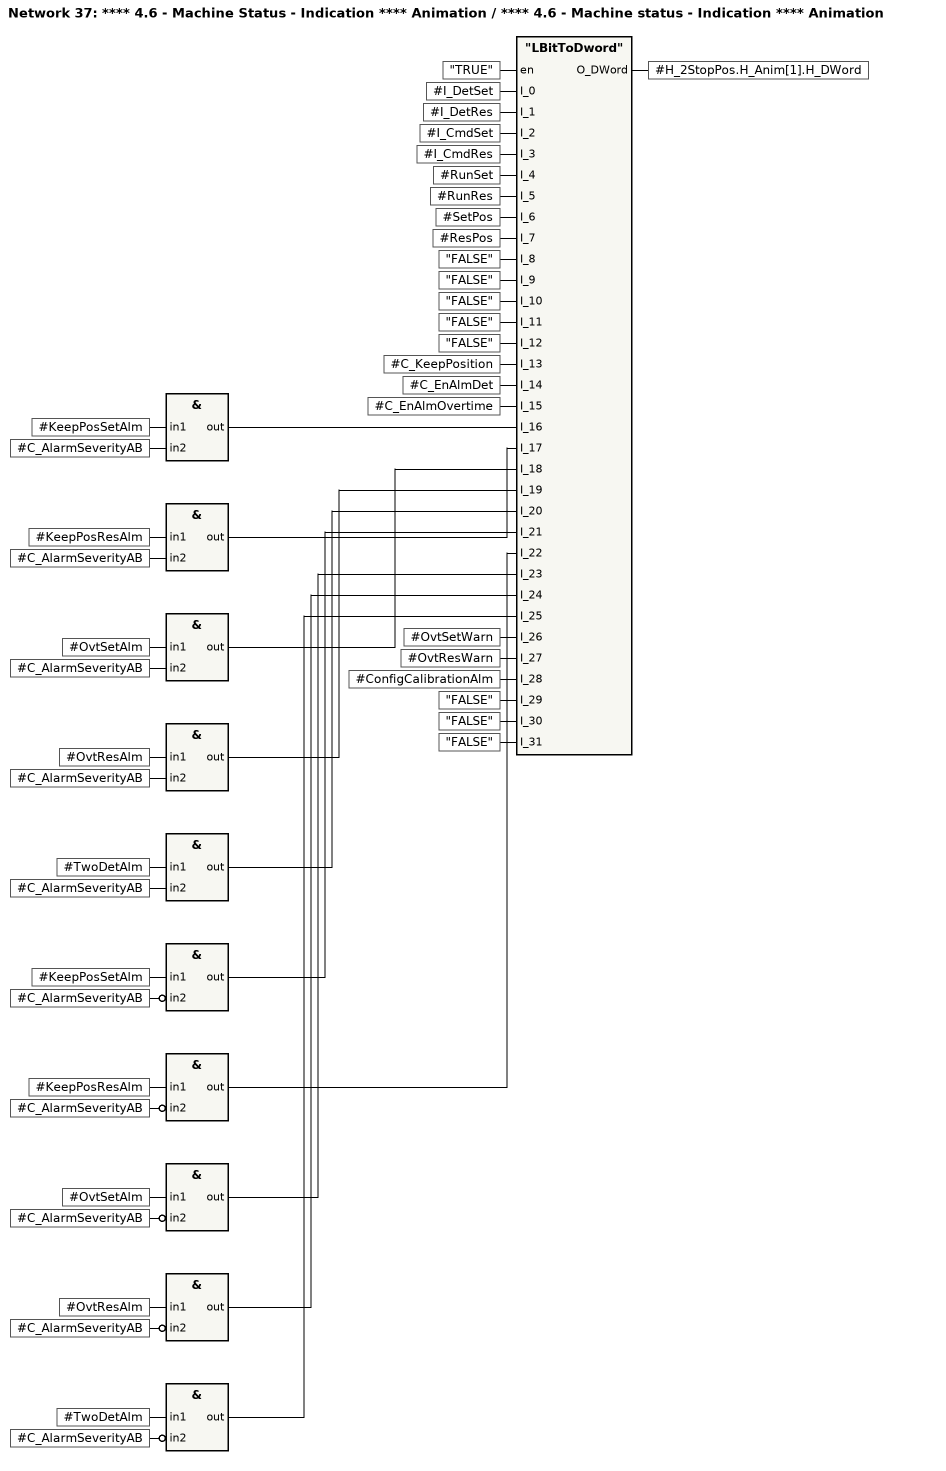
   IF "TRUE" THEN
       "LBitToDword"(I_0 := #I_DetSet,
                     I_1 := #I_DetRes,
                     I_2 := #I_CmdSet,
                     I_3 := #I_CmdRes,
                     I_4 := #RunSet,
                     I_5 := #RunRes,
                     I_6 := #SetPos,
                     I_7 := #ResPos,
                     I_8 := "FALSE",
                     I_9 := "FALSE",
                     I_10 := "FALSE",
                     I_11 := "FALSE",
                     I_12 := "FALSE",
                     I_13 := #C_KeepPosition,
                     I_14 := #C_EnAlmDet,
                     I_15 := #C_EnAlmOvertime,
                     I_16 := #KeepPosSetAlm AND #C_AlarmSeverityAB,
                     I_17 := #KeepPosResAlm AND #C_AlarmSeverityAB,
                     I_18 := #OvtSetAlm AND #C_AlarmSeverityAB,
                     I_19 := #OvtResAlm AND #C_AlarmSeverityAB,
                     I_20 := #TwoDetAlm AND #C_AlarmSeverityAB,
                     I_21 := #KeepPosSetAlm AND NOT #C_AlarmSeverityAB,
                     I_22 := #KeepPosResAlm AND NOT #C_AlarmSeverityAB,
                     I_23 := #OvtSetAlm AND NOT #C_AlarmSeverityAB,
                     I_24 := #OvtResAlm AND NOT #C_AlarmSeverityAB,
                     I_25 := #TwoDetAlm AND NOT #C_AlarmSeverityAB,
                     I_26 := #OvtSetWarn,
                     I_27 := #OvtResWarn,
                     I_28 := #ConfigCalibrationAlm,
                     I_29 := "FALSE",
                     I_30 := "FALSE",
                     I_31 := "FALSE",
                     O_DWord => #H_2StopPos.H_Anim[1].H_DWord);
   END_IF;
END_REGION

REGION Network 38: **** 4.6 - Machine status - Indication **** Animation
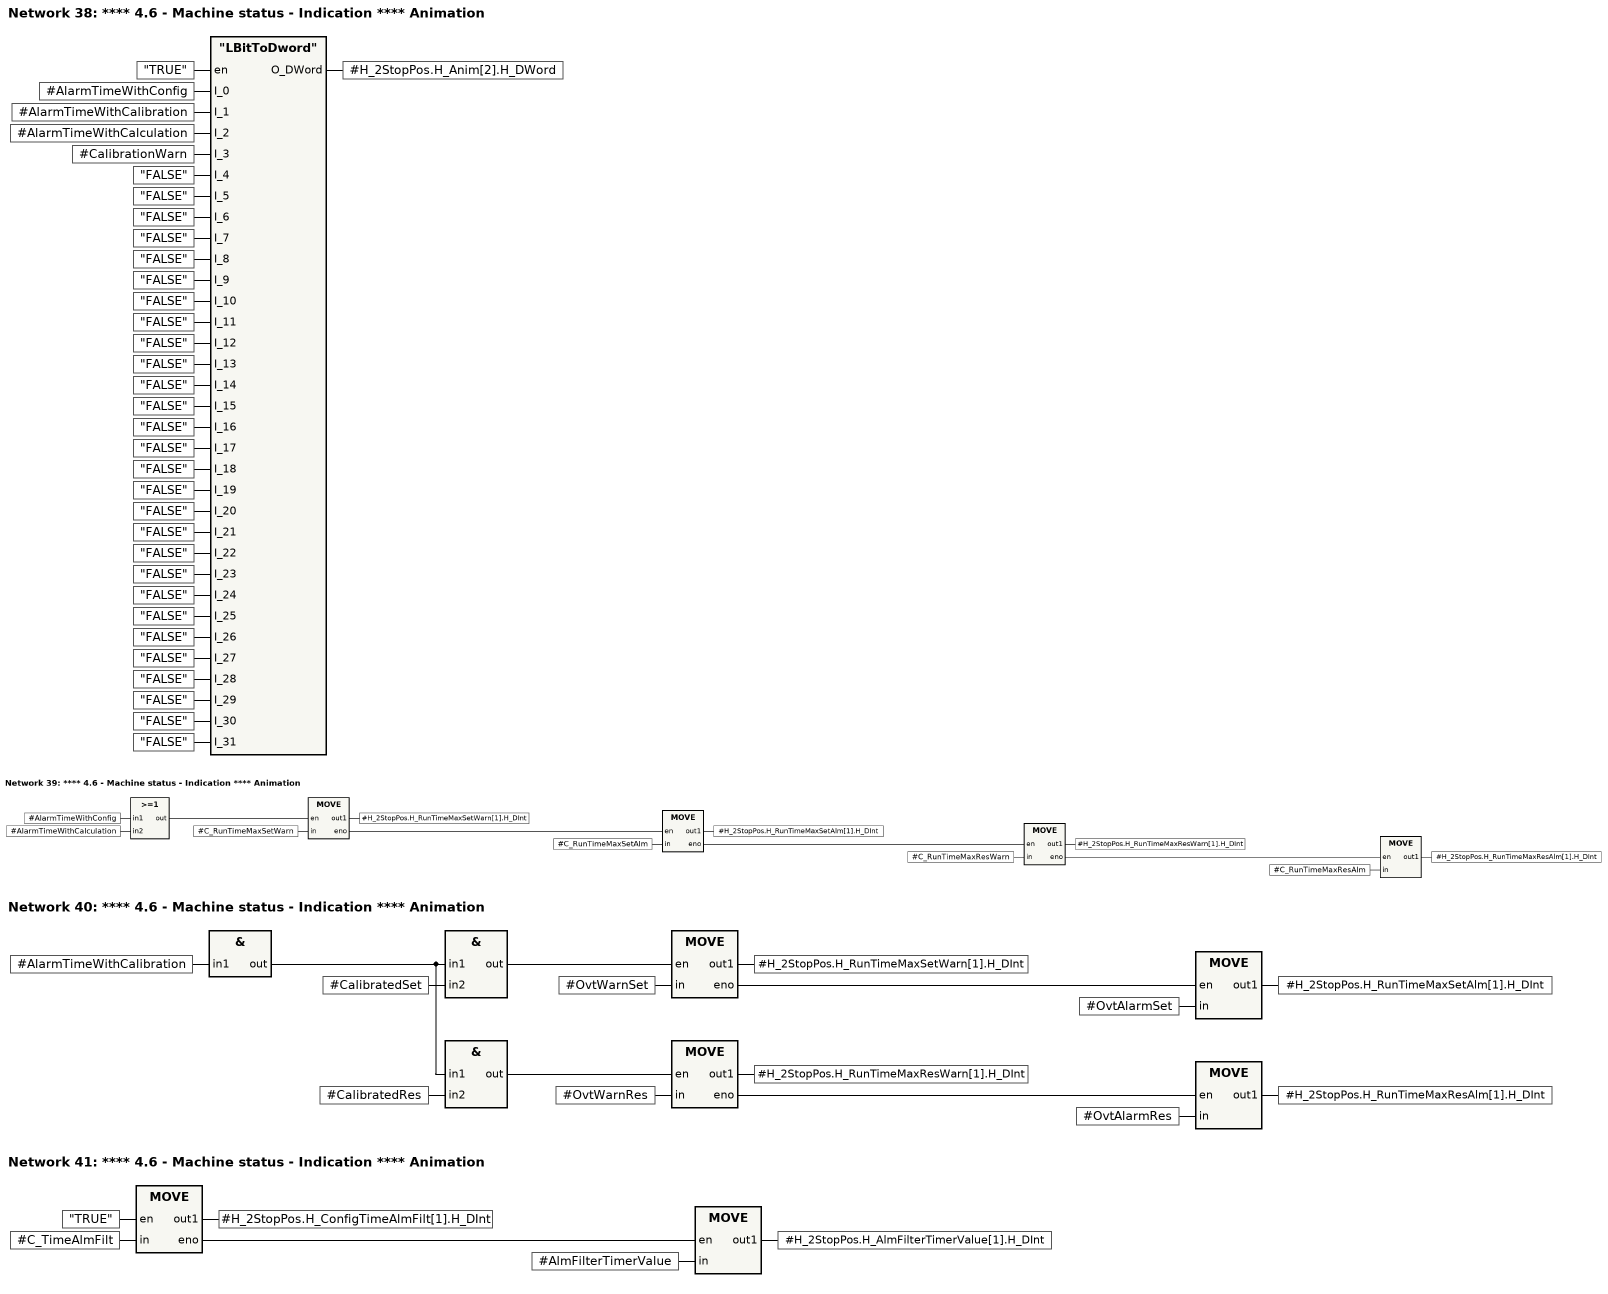
   IF "TRUE" THEN
       "LBitToDword"(I_0 := #AlarmTimeWithConfig,
                     I_1 := #AlarmTimeWithCalibration,
                     I_2 := #AlarmTimeWithCalculation,
                     I_3 := #CalibrationWarn,
                     I_4 := "FALSE",
                     I_5 := "FALSE",
                     I_6 := "FALSE",
                     I_7 := "FALSE",
                     I_8 := "FALSE",
                     I_9 := "FALSE",
                     I_10 := "FALSE",
                     I_11 := "FALSE",
                     I_12 := "FALSE",
                     I_13 := "FALSE",
                     I_14 := "FALSE",
                     I_15 := "FALSE",
                     I_16 := "FALSE",
                     I_17 := "FALSE",
                     I_18 := "FALSE",
                     I_19 := "FALSE",
                     I_20 := "FALSE",
                     I_21 := "FALSE",
                     I_22 := "FALSE",
                     I_23 := "FALSE",
                     I_24 := "FALSE",
                     I_25 := "FALSE",
                     I_26 := "FALSE",
                     I_27 := "FALSE",
                     I_28 := "FALSE",
                     I_29 := "FALSE",
                     I_30 := "FALSE",
                     I_31 := "FALSE",
                     O_DWord => #H_2StopPos.H_Anim[2].H_DWord);
   END_IF;
END_REGION

REGION Network 39: **** 4.6 - Machine status - Indication **** Animation
   IF #AlarmTimeWithConfig OR #AlarmTimeWithCalculation THEN
       #H_2StopPos.H_RunTimeMaxSetWarn[1].H_DInt := #C_RunTimeMaxSetWarn;
       #H_2StopPos.H_RunTimeMaxSetAlm[1].H_DInt := #C_RunTimeMaxSetAlm;
       #H_2StopPos.H_RunTimeMaxResWarn[1].H_DInt := #C_RunTimeMaxResWarn;
       #H_2StopPos.H_RunTimeMaxResAlm[1].H_DInt := #C_RunTimeMaxResAlm;
   END_IF;
END_REGION

REGION Network 40: **** 4.6 - Machine status - Indication **** Animation
   IF #AlarmTimeWithCalibration AND #CalibratedSet THEN
       #H_2StopPos.H_RunTimeMaxSetWarn[1].H_DInt := #OvtWarnSet;
       #H_2StopPos.H_RunTimeMaxSetAlm[1].H_DInt := #OvtAlarmSet;
   END_IF;
   IF #AlarmTimeWithCalibration AND #CalibratedRes THEN
       #H_2StopPos.H_RunTimeMaxResWarn[1].H_DInt := #OvtWarnRes;
       #H_2StopPos.H_RunTimeMaxResAlm[1].H_DInt := #OvtAlarmRes;
   END_IF;
END_REGION

REGION Network 41: **** 4.6 - Machine status - Indication **** Animation
   IF "TRUE" THEN
       #H_2StopPos.H_ConfigTimeAlmFilt[1].H_DInt := #C_TimeAlmFilt;
       #H_2StopPos.H_AlmFilterTimerValue[1].H_DInt := #AlmFilterTimerValue;
   END_IF;
END_REGION

REGION Network 42: **** 5.2 - Equations - Flow Equations **** Set Position
   // Set Position
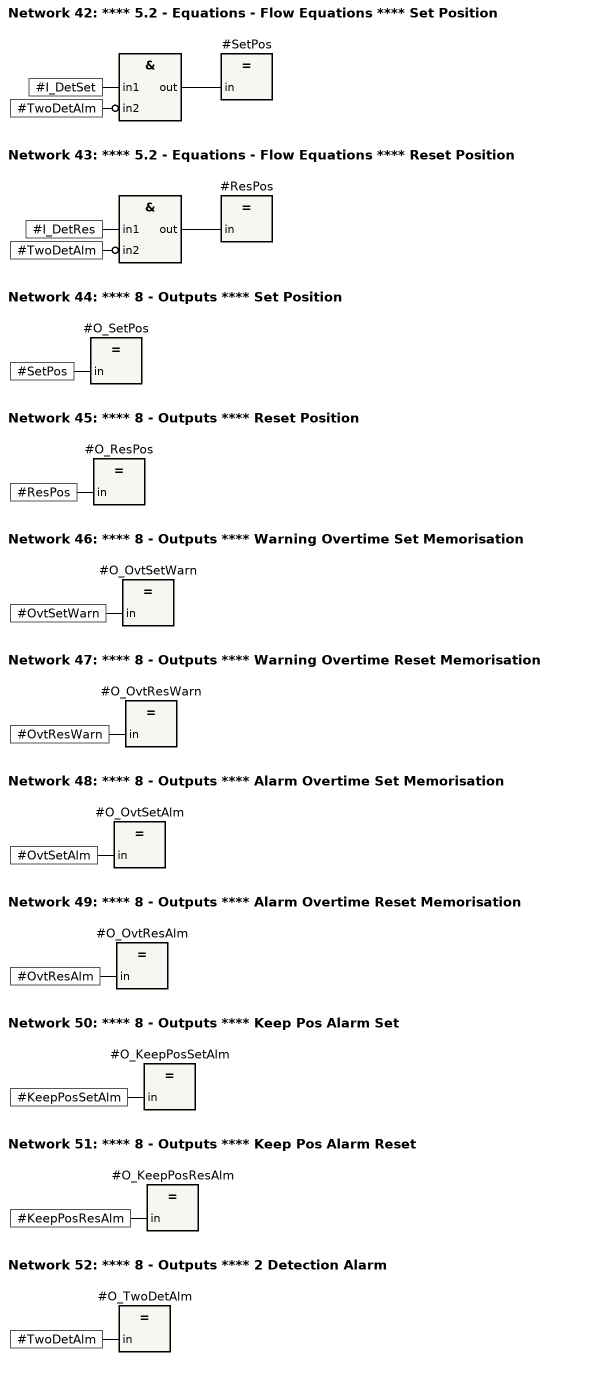
   #SetPos := #I_DetSet AND NOT #TwoDetAlm;
END_REGION

REGION Network 43: **** 5.2 - Equations - Flow Equations **** Reset Position
   // Reset  Position
   #ResPos := #I_DetRes AND NOT #TwoDetAlm;
END_REGION

REGION Network 44: **** 8 - Outputs **** Set Position
   // Set Position
   #O_SetPos := #SetPos;
END_REGION

REGION Network 45: **** 8 - Outputs **** Reset Position
   // Reset  Position
   #O_ResPos := #ResPos;
END_REGION

REGION Network 46: **** 8 - Outputs **** Warning Overtime Set Memorisation
   // Warning Overtime Set Memorisation
   #O_OvtSetWarn := #OvtSetWarn;
END_REGION

REGION Network 47: **** 8 - Outputs **** Warning Overtime Reset Memorisation
   // Warning Overtime Reset  Memorisation
   #O_OvtResWarn := #OvtResWarn;
END_REGION

REGION Network 48: **** 8 - Outputs **** Alarm Overtime Set Memorisation
   // Alarm Overtime Set Memorisation
   #O_OvtSetAlm := #OvtSetAlm;
END_REGION

REGION Network 49: **** 8 - Outputs **** Alarm Overtime Reset Memorisation
   // Alarm Overtime Reset  Memorisation
   #O_OvtResAlm := #OvtResAlm;
END_REGION

REGION Network 50: **** 8 - Outputs **** Keep Pos Alarm Set
   // Keep Pos Alarm Set
   #O_KeepPosSetAlm := #KeepPosSetAlm;
END_REGION

REGION Network 51: **** 8 - Outputs **** Keep Pos Alarm Reset
   // Keep Pos Alarm Reset
   #O_KeepPosResAlm := #KeepPosResAlm;
END_REGION

REGION Network 52: **** 8 - Outputs **** 2 Detection Alarm
   // 2 Detection Alarm
   #O_TwoDetAlm := #TwoDetAlm;
END_REGION

REGION Network 53: **** 8 - Outputs **** Config/Calibration Alarm
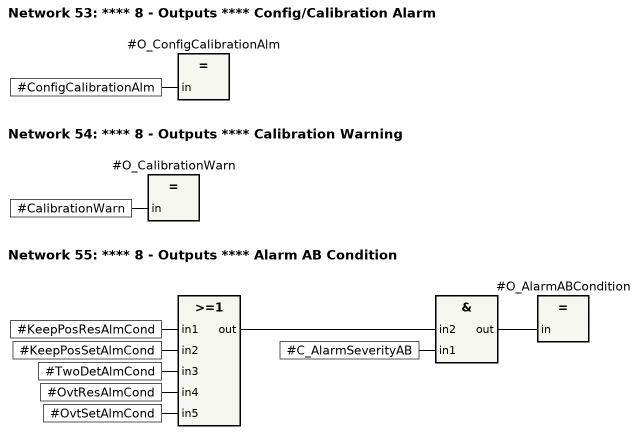
   #O_ConfigCalibrationAlm := #ConfigCalibrationAlm;
END_REGION

REGION Network 54: **** 8 - Outputs **** Calibration Warning
   #O_CalibrationWarn := #CalibrationWarn;
END_REGION

REGION Network 55: **** 8 - Outputs **** Alarm AB Condition
   // Alarm AB Condition
   #O_AlarmABCondition := (#KeepPosResAlmCond OR #KeepPosSetAlmCond OR #TwoDetAlmCond OR #OvtResAlmCond OR #OvtSetAlmCond) AND #C_AlarmSeverityAB;
END_REGION
END_FUNCTION_BLOCK
